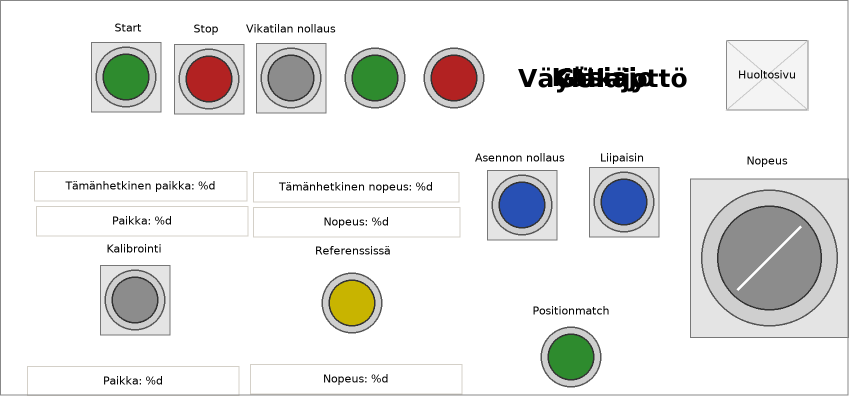
VISUALIZATION Visualization  // 849x396, background image ImagePool.beksu
    PushSwitch (91,42 70x70), variable: GVL.startGUI, behaviour: TAP, style: Switch-PushSwitch-Green
    PushSwitch (174,44 70x70), variable: GVL.stopGUI, behaviour: TAP, style: Switch-PushSwitch-Red
    PushSwitch (256,43 70x70), variable: GVL.resetGUI, behaviour: TAP, style: Switch-PushSwitch-Gray
    Lamp1 (340,43 70x70), variable: GVL.systemOnLight, style: Lamp-Lamp1-Green
    Label (526,63 150x30), "GUIajo", invisible if: control.driverMode2
    Label (528,62 150x30), "Käsiajo", invisible if: control.driverMode1
    Label (503,63 200x30), "Väyläkäyttö", invisible if: control.driverMode3
    Lamp1 (419,43 70x70), variable: GVL.safetyOkLight, style: Lamp-Lamp1-Red
    Textfield (36,206 212x30), "Paikka: %d", text variable: motor.stepperValue, invisible if: control.invisibleGUI
        OnMouseDown: write the text variable via Default
    Textfield (253,207 207x30), "Nopeus: %d", text variable: motor.stepperSpeedGUI, invisible if: control.invisibleGUI
    Textfield (34,171 213x30), "Tämänhetkinen paikka: %d", text variable: motor.currentStepperPosition
    Textfield (253,172 206x30), "Tämänhetkinen nopeus: %d", text variable: motor.CurrentStepperSpeed
    PushSwitch (487,170 70x70), variable: GVL.asemannollausGUI, invisible if: control.invisibleGUI, behaviour: TAP, style: Switch-PushSwitch-Blue
    Label (445,143 150x30), "Asennon nollaus", invisible if: control.invisibleGUI
    Label (216,14 150x30), "Vikatilan nollaus"
    Label (131,14 150x30), "Stop"
    Label (53,13 150x30), "Start"
    PushSwitch (589,167 70x70), variable: GVL.triggerGUI, behaviour: TAP, style: Switch-PushSwitch-Blue
    Label (547,143 150x30), "Liipaisin"
    PushSwitch (100,265 70x70), variable: motor.calibrationBtn, invisible if: control.visibleGUI, behaviour: TAP, style: Switch-PushSwitch-Gray
    Label (59,234 150x30), "Kalibrointi", invisible if: control.visibleGUI
    Lamp1 (317,268 70x70), variable: motor.onReferenceVar, invisible if: control.visibleGUI, style: Lamp-Lamp1-Yellow
    Label (278,236 150x30), "Referenssissä", invisible if: control.visibleGUI
    Label (692,146 150x30), "Nopeus", invisible if: control.invisibleGUI
    Image (726,40 82x70), "Huoltosivu", image: VisuDialogs.ImagePoolDialogs.FileOpen
        OnMouseClick: change screen: Huoltosivu
    Textfield (250,364 212x30), "Nopeus: %d", text variable: motor.stepperSpeedVay, invisible if: control.visibleGUI
        OnMouseDown: write the text variable via Default
    Textfield (27,366 212x30), "Paikka: %d", text variable: motor.stepperValueVay, invisible if: control.visibleGUI
        OnMouseDown: write the text variable via Default
    Potentiometer360 (690,177 159x162), variable: motor.stepperSpeedGUI, style: Potentiometer-Potentiometer360-Gray, scale format: %.1f, scale 0..100
        p2431819421: Outside
    Lamp1 (536,322 70x70), variable: motor.positionMatch, invisible if: control.visibleGUI, style: Lamp-Lamp1-Green
    Label (496,296 150x30), "Positionmatch", invisible if: control.visibleGUI
END_VISUALIZATION

(* stored: Version 1.1.0.1, ProductVersion 3.1.4024.11
   Visu Visualization: Id {45ca7430-5d9c-404d-a6c0-2d552295d7a1} *)
